TYPE STATE:
    STRUCT
        curTime: LREAL;
        dvar_M_a AT %Q*: enum_E;
    END_STRUCT
END_TYPE

(* stored: ProductVersion 3.1.0.18, Version 1.1.0.1 *)
